PROGRAM UnitTests
VAR
	el2574PixelReader_TestSuite : EL2574PixelReader_TestSuite;
END_VAR

TcUnit.RUN();

END_PROGRAM

(* stored: Version 1.1.0.1, ProductVersion 3.1.4024.13
   POU UnitTests: Id {fae0dbda-b8b2-485e-99f6-b0e512bdb931}, SpecialFunc None *)
